TYPE ST_Identity_PK2_OUT2 :
STRUCT
	ID	:STRING;
	ReadQuality:STRING;
END_STRUCT
END_TYPE

(* stored: Version 1.1.0.1, ProductVersion 3.1.4024.13
   DUT ST_Identity_PK2_OUT2: Id {bbbec238-a00e-4145-8310-208c6233e710} *)
